PROGRAM MAIN
VAR
	ctrl: ST_Ctrl;
	status:ST_Status;
	dateiname:STRING:='C:\Temp\Beispielprojekt.pdf';
	
	//Digital I/O
	ATI_input1 AT%I* : BOOL;
	ATI_input2 AT%I* : BOOL;
	
	ATQ_output1 AT%Q* : BOOL;
	ATQ_output2 AT%Q* : BOOL;


	szeit_on:STRING:='500';
	tzeit_on:TIME;
	szeit_off:STRING:='500';
	tzeit_off:TIME;
	
	auswahl_index: INT;
	auswahl : ARRAY[0..2] OF STRING:=['Ein', 'Aus', 'PWM'];
	
	fbpwm: FB_PWM;
	
END_VAR

PRG_PDF(ctrl:=ctrl ,dateiname:=dateiname, status=>status );

//komentar in testverzweigung hinzugefügt

CASE auswahl_index OF
	0: //Ein
		ATQ_output1:=TRUE;
		ATQ_output2:=TRUE;
	1: // Aus
		ATQ_output1:=FALSE;
		ATQ_output2:=FALSE;
		
	2: //PWM	
		tzeit_on:=FUN_String_to_Time(text:=szeit_on);
		tzeit_off:=FUN_String_to_Time(text:=szeit_off);
		fbpwm(tHightime:=tzeit_on, tLowtime:=tzeit_off);
		ATQ_output2:=fbpwm.output;
	ELSE
		;
END_CASE

//in Testverzweigung 1 hinzugefügt
//Kommentar
//kommentar 2

END_PROGRAM

(* stored: Version 1.1.0.1, ProductVersion 3.1.4020.12
   POU MAIN: Id {eb642d55-1955-4dfb-b308-8e501845e6ed}, SpecialFunc None *)
